Universal Robots PolyScope program: From_home_to_spoon.urp

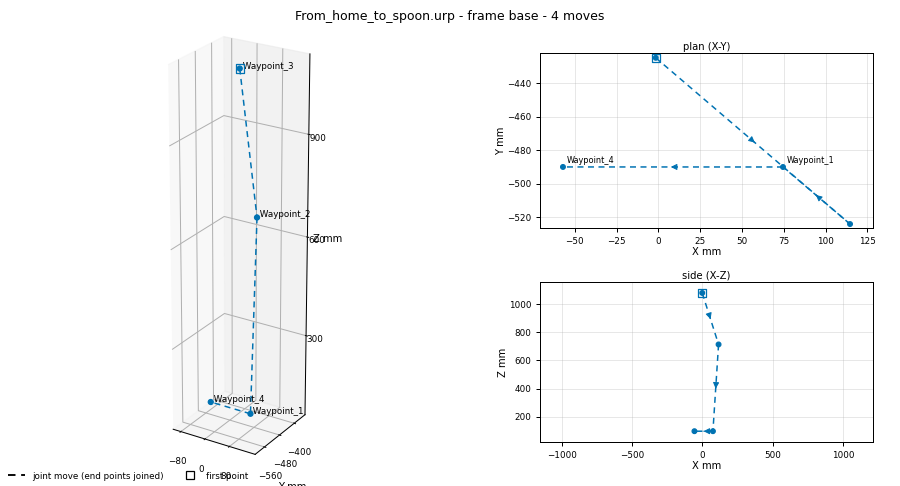
[picture p0: tool path of From_home_to_spoon.urp in frame base, 4 of 4 moves have a stored position in this frame; points joined in program order, loops and branches not executed]
Program From_home_to_spoon (installation=default directory=/programs/Matcha createdIn=5.12.6.1102099 lastSavedIn=5.12.6.1102099 robotSerialNumber=20215500597)
Calibrated DH parameters: a=[0.000193, -0.066673, -0.391568, -0.000012, 0.00005, 0]; d=[0.162643, -472.05677, 465.132521, 7.058239, 0.099746, 0.099582]; alpha=[1.571116, 0.00089, 0.003862, 1.569269, -1.569248, 0]; deltaTheta=[0, -1.413394, 7.628392, 0.068187, 0, -0.000001]
Robot Program (runOnlyOnce=true)
  MoveJ speed 60 deg/s, acceleration 80 deg/s^2 (useActiveTCP=true) feature=Base
    Waypoint Waypoint_3: TCP in base x=-1.543 y=-424.817 z=1080.554 mm, rx=-0.0044 ry=-2.2185 rz=2.2204 rad; joints [0.001, -90, 0.002, -90.002, 0.001, -0.002] deg; TCP offset x=0 y=0 z=191.5 mm, rx=0 ry=0 rz=0 rad
    Waypoint Waypoint_2: TCP in base x=114.633 y=-524.214 z=714.145 mm, rx=1.8679 ry=-0.6918 rz=1.9311 rad; joints [50.058, -96.38, 92.167, -171.188, 4.73, -89.222] deg
    Waypoint Waypoint_1: TCP in base x=74.541 y=-490.092 z=96.965 mm, rx=-0.014 ry=1.5917 rz=-0.0243 rad; joints [51.586, -52.596, 101.87, -51.014, -37.915, -90.057] deg
    Waypoint Waypoint_4: TCP in base x=-57.022 y=-490.067 z=96.967 mm, rx=-0.014 ry=1.5917 rz=-0.0243 rad; joints [41.637, -46.217, 88.999, -44.212, -47.882, -90.493] deg
